INTERFACE I_FileHandler EXTENDS I_Component, I_Cyclic, I_TaskResult, I_TaskResult, I_Resettable

METHOD ClearDocument
VAR_INPUT
END_VAR
END_METHOD

PROPERTY Datatype : T_MaxString
SET
END_SET
END_PROPERTY

METHOD LoadFile
END_METHOD

PROPERTY nData : UDINT
SET
END_SET
END_PROPERTY

PROPERTY PUBLIC Path : T_MaxString
GET
END_GET
SET
END_SET
END_PROPERTY

PROPERTY pData : PVOID
SET
END_SET
END_PROPERTY

METHOD ReadSymbol
END_METHOD

METHOD SaveFile
END_METHOD

PROPERTY SymbolName : T_MaxString
SET
END_SET
END_PROPERTY

PROPERTY Timeout : TIME
SET
END_SET
END_PROPERTY

METHOD UpdateSymbol
END_METHOD

END_INTERFACE

(* stored: Version 1.1.0.1, ProductVersion 3.1.4026.18
   Itf I_FileHandler: Id {55011597-79d0-4949-85e2-2be0ab2b934d}
   Method ClearDocument: Id {8fb4a3e4-6d56-0aae-1c44-81e342d914a2}
   Property Datatype: Id {a0521760-68d0-4d0f-a9e5-f3f3fe686ce0}
   Set Set: Id {2475b506-8cb8-4f10-8139-f57c90ea8e01}
   Method LoadFile: Id {3ab11060-e413-4c53-a193-f19323c61c38}
   Property nData: Id {4ef7b631-7d6c-4586-bd16-b2a5d96207f6}
   Set Set: Id {5674a16e-4cf0-4f05-97d1-7f124fa057f6}
   Property Path: Id {493c8d8b-b87e-478e-a1a6-c7ad2156433a}
   Get Get: Id {a6759574-5ef5-45a1-b11f-c3268fd3a4ae}
   Set Set: Id {b38783df-9042-493c-873b-9f9bdd19f7e6}
   Property pData: Id {630e1e7d-adf3-4054-9b32-3935a30b990a}
   Set Set: Id {9ac28e23-ffe4-4a98-ba1c-f05319aa474c}
   Method ReadSymbol: Id {02f0cf69-dcff-4c9a-8129-b397d230c959}
   Method SaveFile: Id {99ad8ae3-4840-423d-afaf-d359726ad74f}
   Property SymbolName: Id {1128767d-b7e7-4468-8549-49cc2ac2a464}
   Set Set: Id {ba00c0e0-f437-40a1-a4d5-41439f1a9b07}
   Property Timeout: Id {d36ed3da-17f1-0c1f-01c1-ab686683753c}
   Set Set: Id {34384024-0a9b-0303-3c3b-8ca68d115331}
   Method UpdateSymbol: Id {d8d2a82b-5421-44b8-9fab-ead5518be454} *)
